(* CoDeSys 2.3.9.40 project: doz_qizil.pro *)
(* Libraries: STANDARD.LIB 4.10.05 11:14:46, IECSFC.LIB 13.4.06 15:51:28, SYSLIBTIME.LIB 20.2.06 13:31:16, SYSTASKINFO.LIB 20.2.06 13:31:38, ANALYZATION.LIB 5.10.99 09:05:06, SYSLIBCALLBACK.LIB 20.2.06 13:31:08, Util.lib 18.5.10 15:14:28 *)

(* PLC configuration (modules and I/O channels)
Fast discrete inputs [I_SIMPLE_INPUT] node 0, in %IB0 out %QB0 {Filtrationtime = 10}
  speedImpuls1 AT %IX0.0 [BitInput] Discrete input 1
  speedImpuls2 AT %IX0.1 [BitInput] Discrete input 2
  speedImpuls3 AT %IX0.2 [BitInput] Discrete input 3
  speedImpuls4 AT %IX0.3 [BitInput] Discrete input 4
AT %IB1.0 [ByteInput] 8 discrete inputs
AT %IB1.1 [ByteInput] 8 discrete inputs
AT %IB1.2 [ByteInput] 8 discrete inputs
AT %IB1.3 [ByteInput] 8 discrete inputs
Fast discrete outputs [OWEN_ID570] node 2, in %IB2 out %QB2 {SafeValueBool = FALSE; SafeValueBool = FALSE; SafeValueBool = FALSE; SafeValueBool = FALSE; Visibility = No}
  runChastot1 AT %QX2.0 [BitOutput] Fast discrete output 1
  runChastot2 AT %QX2.1 [BitOutput] Fast discrete output 2
  runChastot3 AT %QX2.2 [BitOutput] Fast discrete output 3
  runChastot4 AT %QX2.3 [BitOutput] Fast discrete output 4
Discrete outputs [ID131] node 3, in %IB3 out %QB3 {SafeValueByte = 0; SafeValueByte = 0; SafeValueByteM = 0; Visibility = No; PinCount = 24}
  AT %QB3.0 [ByteOutput] 8 discrete outputs
  AT %QB3.1 [ByteOutput] 8 discrete outputs
  AT %QB3.2 [ByteOutput] 4 discrete outputs
Special input [ID103] node 4, in %IB4 out %QB4 {Filtrationtime = 1000; PinCount = 1; WatchDogPeriod = 400; PollPeriod = 3000; Visibility = No}
  AT %IX4.0 [BitInput] Special input
Special output [ID104] node 5, in %IB5 out %QB5 {Visibility = No; PinCount = 1}
  AT %QX5.0 [BitOutput] Special output
DCON (Master) [DCON_MASTER_ID452] node 6, in %IB6 out %QB6 {Visibility = No}
  AT %QW6.0 [WordOutput] Last error
  RS-485-1 [COM1_USART] node 0, in %IB6.0 out %QB6.0 {CommunicationSpeed = 57600; Parity = NO PARITY CHECK; BitLength = 8 bits; StopLength = One stop bit; InterfaceType = RS485; FrameOriented = ASCII; Timeout = 0; Visibility = No}
  Universal DCON device [ID2100] node 1, in %IB6.1 out %QB6.1 {ReqFormat = #010[7s]; GoodResponseFormat = [1s]; BadResponseFormat = ?; ServiceTimeout = 150; RequestType = By poll time; PeriodOfService = 100; Visibility = No}
    AT %QW6.1.0 [WordOutput] Status
AT %IB6.1.0.0 [StringInput]
outVolt1 AT %QB6.1.1.0 [StringOutput]
Universal DCON device [ID2100] node 2, in %IB6.2 out %QB6.2 {ReqFormat = #011[7s]; GoodResponseFormat = [1s]; BadResponseFormat = ?; ServiceTimeout = 150; RequestType = By poll time; PeriodOfService = 100; Visibility = No}
  AT %QW6.2.0 [WordOutput] Status
AT %IB6.2.0.0 [StringInput]
outVolt2 AT %QB6.2.1.0 [StringOutput]
Universal DCON device [ID2100] node 3, in %IB6.3 out %QB6.3 {ReqFormat = #012[7s]; GoodResponseFormat = [1s]; BadResponseFormat = ?; ServiceTimeout = 150; RequestType = By poll time; PeriodOfService = 100; Visibility = No}
  AT %QW6.3.0 [WordOutput] Status
AT %IB6.3.0.0 [StringInput]
outVolt3 AT %QB6.3.1.0 [StringOutput]
Universal DCON device [ID2100] node 4, in %IB6.4 out %QB6.4 {ReqFormat = #013[7s]; GoodResponseFormat = [1s]; BadResponseFormat = ?; ServiceTimeout = 150; RequestType = By poll time; PeriodOfService = 100; Visibility = No}
  AT %QW6.4.0 [WordOutput] Status
AT %IB6.4.0.0 [StringInput]
outVolt4 AT %QB6.4.1.0 [StringOutput]
Universal DCON device [ID2100] node 5, in %IB6.5 out %QB6.5 {ReqFormat = #021; GoodResponseFormat = >[7f]; BadResponseFormat = ?; ServiceTimeout = 150; RequestType = By poll time; PeriodOfService = 100; Visibility = No}
  AT %QW6.5.0 [WordOutput] Status
dozWeight1 AT %ID6.5.0.0 [FloatInput]
Universal DCON device [ID2100] node 6, in %IB6.6 out %QB6.6 {ReqFormat = #022; GoodResponseFormat = >[7f]; BadResponseFormat = ?; ServiceTimeout = 150; RequestType = By poll time; PeriodOfService = 100; Visibility = No}
  AT %QW6.6.0 [WordOutput] Status
dozWeight2 AT %ID6.6.0.0 [FloatInput]
Universal DCON device [ID2100] node 7, in %IB6.7 out %QB6.7 {ReqFormat = #023; GoodResponseFormat = >[7f]; BadResponseFormat = ?; ServiceTimeout = 150; RequestType = By poll time; PeriodOfService = 100; Visibility = No}
  AT %QW6.7.0 [WordOutput] Status
dozWeight3 AT %ID6.7.0.0 [FloatInput]
Universal DCON device [ID2100] node 8, in %IB6.8 out %QB6.8 {ReqFormat = #024; GoodResponseFormat = >[7f]; BadResponseFormat = ?; ServiceTimeout = 150; RequestType = By poll time; PeriodOfService = 100; Visibility = No}
  AT %QW6.8.0 [WordOutput] Status
dozWeight4 AT %ID6.8.0.0 [FloatInput]
RS-232 [COM2_USART] node 0, in %IB7.0.0 out %QB7.0.0 {CommunicationSpeed = 57600; Parity = NO PARITY CHECK; BitLength = 8 bits; StopLength = One stop bit; InterfaceType = RS232; FrameOriented = RTU; Timeout = 0; Visibility = No}
Debug RS-232 [DEBUG_USART] node 1, in %IB7.0.1 out %QB7.0.1 {CommunicationSpeed = 57600; Parity = NO PARITY CHECK; BitLength = 8 bits; StopLength = One stop bit; InterfaceType = RS232; FrameOriented = RTU; Timeout = 0; Visibility = No}
AT %QD7.1.0 [FloatOutput]
AT %QD7.2.0 [FloatOutput]
AT %QD7.3.0 [FloatOutput]
AT %QD7.4.0 [FloatOutput]
AT %QD7.5.0 [FloatOutput]
AT %QD7.6.0 [FloatOutput]
AT %QD7.7.0 [FloatOutput]
AT %QD7.8.0 [FloatOutput]
AT %QD7.9.0 [FloatOutput]
AT %QD7.10.0 [FloatOutput]
AT %QD7.11.0 [FloatOutput]
AT %QD7.12.0 [FloatOutput]
AT %QD7.13.0 [FloatOutput]
AT %QD7.14.0 [FloatOutput]
AT %QD7.15.0 [FloatOutput]
AT %QD7.16.0 [FloatOutput]
AT %QD7.17.0 [FloatOutput]
AT %QD7.18.0 [FloatOutput]
AT %QD7.19.0 [FloatOutput]
AT %QD7.20.0 [FloatOutput]
AT %QD7.21.0 [FloatOutput]
AT %QD7.22.0 [FloatOutput]
AT %QD7.23.0 [FloatOutput]
AT %QD7.24.0 [FloatOutput]
AT %QD7.25.0 [FloatOutput]
AT %QD7.26.0 [FloatOutput]
AT %QD7.27.0 [FloatOutput]
AT %QD7.28.0 [FloatOutput]
AT %QD7.29.0 [FloatOutput]
AT %QD7.30.0 [FloatOutput]
AT %QD7.31.0 [FloatOutput]
AT %QD7.32.0 [FloatOutput]
AT %QD7.33.0 [FloatOutput]
AT %QD7.34.0 [FloatOutput]
AT %QD7.35.0 [FloatOutput]
AT %QD7.36.0 [FloatOutput]
AT %QD7.37.0 [FloatOutput]
AT %QD7.38.0 [FloatOutput]
AT %QD7.39.0 [FloatOutput]
AT %QD7.40.0 [FloatOutput]
AT %QD7.41.0 [FloatOutput]
AT %QW7.42.0 [WordOutput]
AT %QW7.43.0 [WordOutput]
AT %QW7.44.0 [WordOutput]
AT %QW7.45.0 [WordOutput]
8 bits [8Bit] node 46, in %IB7.46 out %QB7.46
  AT %QB7.46.0 [ByteOutput]
8 bits [8Bit] node 47, in %IB7.47 out %QB7.47
  AT %QB7.47.0 [ByteOutput]
8 bits [8Bit] node 48, in %IB7.48 out %QB7.48
  AT %QB7.48.0 [ByteOutput]
  AT %QB7.49.0 [ByteOutput]
Float [Float] node 50, in %IB7.50 out %QB7.50
  AT %QD7.50.0 [FloatOutput]
  AT %QD7.51.0 [FloatOutput]
  AT %QD7.52.0 [FloatOutput]
  AT %QD7.53.0 [FloatOutput]
  AT %QD7.54.0 [FloatOutput]
  AT %QD7.55.0 [FloatOutput]
  AT %QD7.56.0 [FloatOutput]
  AT %QD7.57.0 [FloatOutput]
  AT %QD7.58.0 [FloatOutput]
  AT %QD7.59.0 [FloatOutput]
Float [Float] node 60, in %IB7.60 out %QB7.60
  AT %QD7.60.0 [FloatOutput]
2 byte [Register] node 61, in %IB7.61 out %QB7.61
  year AT %QW7.61.0 [WordOutput]
2 byte [Register] node 62, in %IB7.62 out %QB7.62
  month AT %QW7.62.0 [WordOutput]
2 byte [Register] node 63, in %IB7.63 out %QB7.63
  day AT %QW7.63.0 [WordOutput]
2 byte [Register] node 64, in %IB7.64 out %QB7.64
  hour AT %QW7.64.0 [WordOutput]
2 byte [Register] node 65, in %IB7.65 out %QB7.65
  minute AT %QW7.65.0 [WordOutput]
2 byte [Register] node 66, in %IB7.66 out %QB7.66
  sekund AT %QW7.66.0 [WordOutput]
2 byte [Register] node 67, in %IB7.67 out %QB7.67
  taskDozSpeed1 AT %QW7.67.0 [WordOutput]
2 byte [Register] node 68, in %IB7.68 out %QB7.68
  taskDozSpeed2 AT %QW7.68.0 [WordOutput]
2 byte [Register] node 69, in %IB7.69 out %QB7.69
  taskDozSpeed3 AT %QW7.69.0 [WordOutput]
2 byte [Register] node 70, in %IB7.70 out %QB7.70
  taskDozSpeed4 AT %QW7.70.0 [WordOutput]
  workMode AT %QW7.71.0 [WordOutput]
  AT %QW7.72.0 [WordOutput]
taraSpeedDoz1 AT %QD7.73.0 [FloatOutput]
taraSpeedDoz2 AT %QD7.74.0 [FloatOutput]
taraSpeedDoz3 AT %QD7.75.0 [FloatOutput]
taraSpeedDoz4 AT %QD7.76.0 [FloatOutput]
taraVesDoz1 AT %QD7.77.0 [FloatOutput]
taraVesDoz2 AT %QD7.78.0 [FloatOutput]
taraVesDoz3 AT %QD7.79.0 [FloatOutput]
taraVesDoz4 AT %QD7.80.0 [FloatOutput]
AT %QB7.81.0 [ByteOutput]
AT %QB7.82.0 [ByteOutput]
AT %QB7.83.0 [ByteOutput]
AT %QB7.84.0 [ByteOutput]
AT %QB7.85.0 [ByteOutput]
AT %QB7.86.0 [ByteOutput]
AT %QB7.87.0 [ByteOutput]
AT %QB7.88.0 [ByteOutput]
ModBus (Master) [MODBUS_MASTER_ID450] node 8, in %IB8 out %QB8 {Visibility = No}
  AT %QD8.0 [DWordOutput] Last address
  AT %QW8.1 [WordOutput] Last error
  RS-485-2 [COM3_USART] node 0, in %IB8.0 out %QB8.0 {CommunicationSpeed = 11520; Parity = NO PARITY CHECK; BitLength = 8 bits; StopLength = One stop bit; InterfaceType = RS485; FrameOriented = RTU; Timeout = 0; Visibility = No}
AT %QB8.1.0 [ComChannel] Command (0xff - Start)
freqStatus1 AT %IW8.1.0.0 [WordInput]
freqChastot1 AT %IW8.1.1.0 [WordInput]
freqChastotZadan1 AT %IW8.1.2.0 [WordInput]
freqTok1 AT %IW8.1.3.0 [WordInput]
AT %QB8.2.0 [ComChannel] Command (0xff - Start)
freqStatus2 AT %IW8.2.0.0 [WordInput]
freqChastot2 AT %IW8.2.1.0 [WordInput]
freqChastotZadan2 AT %IW8.2.2.0 [WordInput]
freqTok2 AT %IW8.2.3.0 [WordInput]
AT %QB8.3.0 [ComChannel] Command (0xff - Start)
freqStatus3 AT %IW8.3.0.0 [WordInput]
freqChastot3 AT %IW8.3.1.0 [WordInput]
freqChastotZadan3 AT %IW8.3.2.0 [WordInput]
freqTok3 AT %IW8.3.3.0 [WordInput]
AT %QB8.4.0 [ComChannel] Command (0xff - Start)
freqStatus4 AT %IW8.4.0.0 [WordInput]
freqChastot4 AT %IW8.4.1.0 [WordInput]
freqChastotZadan4 AT %IW8.4.2.0 [WordInput]
freqTok4 AT %IW8.4.3.0 [WordInput]
AT %IX9.0 [BitInput] Button Start/Stop
*)

(* Global variable list: Global_Variables *)
VAR_GLOBAL
	currProizDoz1 AT %QD7.1.0 : REAL; (* 0 *)
	currProizDoz2 AT %QD7.2.0 : REAL; (* 2 *)
	currProizDoz3 AT %QD7.3.0 : REAL; (* 4 *)
	currProizDoz4 AT %QD7.4.0 : REAL; (* 6 *)
	currProizDozTotal AT %QD7.58.0 : REAL; (* 104 *)
	(**************************************************)
	taskDozPercent1 AT %QD7.5.0 : REAL; (* 8 *)
	taskDozPercent2 AT %QD7.6.0 : REAL; (* 10 *)
	taskDozPercent3 AT %QD7.7.0 : REAL; (* 12 *)
	taskDozPercent4 AT %QD7.8.0 : REAL; (* 14 *)
	(**************************************************)
	dozCount1 AT %QD7.9.0 : REAL; (* 16 *)
	dozCount2 AT %QD7.10.0 : REAL; (* 18 *)
	dozCount3 AT %QD7.11.0 : REAL; (* 20 *)
	dozCount4 AT %QD7.12.0 : REAL; (* 22 *)
	dozCountTotal AT %QD7.59.0 : REAL; (* 106 *)
	(**************************************************)
	dozSpeed1 AT %QD7.13.0 : REAL; (* 24 *)
	dozSpeed2 AT %QD7.14.0 : REAL; (* 26 *)
	dozSpeed3 AT %QD7.15.0 : REAL; (* 28 *)
	dozSpeed4 AT %QD7.16.0 : REAL; (* 30 *)
	(**************************************************)
	dozMilliVolt1 AT %QD7.17.0 : REAL; (* 32 *)
	dozMilliVolt2 AT %QD7.18.0 : REAL; (* 34 *)
	dozMilliVolt3 AT %QD7.19.0 : REAL; (* 36 *)
	dozMilliVolt4 AT %QD7.20.0 : REAL; (* 38 *)
	(**************************************************)
	chatotTok1 AT %QD7.21.0 : REAL; (* 40 *)
	chatotTok2 AT %QD7.22.0 : REAL; (* 42 *)
	chatotTok3 AT %QD7.23.0 : REAL; (* 44 *)
	chatotTok4 AT %QD7.24.0 : REAL; (* 46 *)
	(**************************************************)
	chatotFreq1 AT %QD7.25.0 : REAL; (* 48 *)
	chatotFreq2 AT %QD7.26.0 : REAL; (* 50 *)
	chatotFreq3 AT %QD7.27.0 : REAL; (* 52 *)
	chatotFreq4 AT %QD7.28.0 : REAL; (* 54 *)
	(**************************************************)
	taskTotal AT %QD7.29.0: REAL;	(* 56 *)
	(**************************************************)
	dozKoefPerVESDoz1 AT %QD7.30.0: REAL;	(* 58 *)
	dozKoefPerVESDoz2 AT %QD7.31.0: REAL;	(* 60 *)
	dozKoefPerVESDoz3 AT %QD7.32.0 : REAL; (* 62 *)
	dozKoefPerVESDoz4 AT %QD7.33.0 : REAL; (* 64 *)
	(**************************************************)
	dozKoefSpeedDoz1 AT %QD7.34.0 : REAL; (* 66 *)
	dozKoefSpeedDoz2 AT %QD7.35.0 : REAL; (* 68 *)
	dozKoefSpeedDoz3 AT %QD7.36.0 : REAL; (* 70 *)
	dozKoefSpeedDoz4 AT %QD7.37.0 : REAL; (* 72 *)
	(**************************************************)
	dozDreyfDoz1 AT %QD7.38.0 : REAL; (* 74 *)
	dozDreyfDoz2 AT %QD7.39.0 : REAL; (* 76 *)
	dozDreyfDoz3 AT %QD7.40.0 : REAL; (* 78 *)
	dozDreyfDoz4 AT %QD7.41.0 : REAL; (* 80 *)
	(**************************************************)
	dozSkolTimeDoz1 AT %QW7.42.0 : WORD; (* 82 *)
	dozSkolTimeDoz2 AT %QW7.43.0 : WORD; (* 83 *)
	dozSkolTimeDoz3 AT %QW7.44.0 : WORD; (* 84 *)
	dozSkolTimeDoz4 AT %QW7.45.0 : WORD; (* 85 *)
	(**************************************************)
	KoefPer1 AT %QX7.46.0.0 : BOOL; (* 0008600 *)
	KoefPer2 AT %QX7.46.0.1 : BOOL; (* 0008601 *)
	KoefPer3 AT %QX7.46.0.2 : BOOL; (* 0008602 *)
	KoefPer4 AT %QX7.46.0.3 : BOOL; (* 0008603 *)
	(**************************************************)
	KoefSpeed1 AT %QX7.46.0.4 : BOOL; (* 0008604 *)
	KoefSpeed2 AT %QX7.46.0.5 : BOOL; (* 0008605 *)
	KoefSpeed3 AT %QX7.46.0.6 : BOOL; (* 0008606 *)
	KoefSpeed4 AT %QX7.46.0.7 : BOOL; (* 0008607 *)
	(**************************************************)
	dreyf1 AT %QX7.47.0.0 : BOOL; (* 0008608 *)
	dreyf2 AT %QX7.47.0.1 : BOOL; (* 0008609 *)
	dreyf3 AT %QX7.47.0.2 : BOOL; (* 0008610 *)
	dreyf4 AT %QX7.47.0.3 : BOOL; (* 0008611 *)
	(**************************************************)
	resetError AT %QX7.47.0.4 : BOOL; (* 0008612 *)
	timeSinxron AT %QX7.47.0.5 : BOOL; (* 0008613 *)
	(**************************************************)
	dozInGroup1 AT %QX7.48.0.0 : BOOL; (* 0008700 *)
	dozInGroup2 AT %QX7.48.0.1 : BOOL; (* 0008701 *)
	dozInGroup3 AT %QX7.48.0.2 : BOOL; (* 0008702 *)
	dozInGroup4 AT %QX7.48.0.3 : BOOL; (* 0008703 *)
	(**************************************************)
	dozWork1 AT %QX7.48.0.4 : BOOL; (* 0008704 *)
	dozWork2 AT %QX7.48.0.5 : BOOL; (* 0008705 *)
	dozWork3 AT %QX7.48.0.6 : BOOL; (* 0008706 *)
	dozWork4 AT %QX7.48.0.7 : BOOL; (* 0008707 *)
	(**************************************************)
	run1 AT %QX7.49.0.0 : BOOL; (* 0008708 *)
	run2 AT %QX7.49.0.1 : BOOL; (* 0008709 *)
	run3 AT %QX7.49.0.2 : BOOL; (* 0008710 *)
	run4 AT %QX7.49.0.3 : BOOL; (* 0008711 *)
	(**************************************************)
	dozWieght1 AT %QD7.50.0 : REAL; (* 88 *)
	dozWieght2 AT %QD7.51.0 : REAL; (* 90 *)
	dozWieght3 AT %QD7.52.0 : REAL; (* 92 *)
	dozWieght4 AT %QD7.53.0 : REAL; (* 94 *)
	(**************************************************)
	taskProizDoz1 AT %QD7.54.0 : REAL; (* 96 *)
	taskProizDoz2 AT %QD7.55.0 : REAL; (* 98 *)
	taskProizDoz3 AT %QD7.56.0 : REAL; (* 100 *)
	taskProizDoz4 AT %QD7.57.0 : REAL; (* 102 *)
	(**************************************************)
	dreyfTaraVes1 : REAL;
	dreyfTaraVes2 : REAL;
	dreyfTaraVes3 : REAL;
	dreyfTaraVes4 : REAL;

END_VAR

(* POU PLC_PRG, ST *)
PROGRAM PLC_PRG
VAR
	temp : WORD;
END_VAR
(*****************************)
translate();
errors();
sinxron();
sirenStart();
sirenStop();
stopCFC();
(*****************************)
IF(temp <> workMode) THEN
	stopCFC();
	temp := workMode;
END_IF;

CASE workMode OF
	11 : taraSpeedModeDoz1();
	12 : taraSpeedModeDoz2();
	13 : taraSpeedModeDoz3();
	14 : taraSpeedModeDoz4();
	21 : taraVesModeDoz1();
	22 : taraVesModeDoz2();
	23 : taraVesModeDoz3();
	24 : taraVesModeDoz4();
ELSE
	 auto ();
END_CASE;
END_PROGRAM

(* POU translate, ST *)
PROGRAM translate
VAR
	count1 : HISOBLAGICH;
	count2 : HISOBLAGICH;
	count3 : HISOBLAGICH;
	count4 : HISOBLAGICH;

	calcWeight1 : CALCWEIGHT;
	calcWeight2 : CALCWEIGHT;
	calcWeight3 : CALCWEIGHT;
	calcWeight4 : CALCWEIGHT;

	filtr1 : ANALOGFILTR;
	filtr2 : ANALOGFILTR;
	filtr3 : ANALOGFILTR;
	filtr4 : ANALOGFILTR;




END_VAR
(**************************************************)
count1(	tezlik := dozSpeed1,
			proizvodMgn := currProizDoz1,
			SUMMA => dozCount1);
count2(tezlik := dozSpeed2,
			proizvodMgn := currProizDoz2,
			SUMMA => dozCount2);
count3(	tezlik := dozSpeed3,
			proizvodMgn := currProizDoz3,
			SUMMA => dozCount3);
count4(tezlik := dozSpeed4,
			proizvodMgn := currProizDoz4,
			SUMMA => dozCount4);
dozSpeed1 := dozKoefSpeedDoz1 * freqChastotZadan1 ;
dozSpeed2 := dozKoefSpeedDoz2 * freqChastotZadan2;
dozSpeed3 := dozKoefSpeedDoz3 * freqChastotZadan3;
dozSpeed4 := dozKoefSpeedDoz4 * freqChastotZadan4;

calcWeight1(dreyfNol := dozDreyfDoz1,
				koeffitsentPeredachaVes := dozKoefPerVESDoz1,
				milliVolt := dozMilliVolt1,
				Ves => dozWieght2);
calcWeight2(dreyfNol := dozDreyfDoz2,
				koeffitsentPeredachaVes := dozKoefPerVESDoz2,
				milliVolt := dozMilliVolt2,
				Ves => dozWieght2);
calcWeight3(dreyfNol := dozDreyfDoz3,
				koeffitsentPeredachaVes := dozKoefPerVESDoz3,
				milliVolt := dozMilliVolt3,
				Ves => dozWieght3);
calcWeight4(dreyfNol := dozDreyfDoz4,
				koeffitsentPeredachaVes := dozKoefPerVESDoz4,
				milliVolt := dozMilliVolt4,
				Ves => dozWieght4);

dozInGroup1 := doz1InGroup;
dozInGroup2 := doz2InGroup;
dozInGroup3 := doz3InGroup;
dozInGroup4 := doz4InGroup;
currProizDozTotal := currProizDoz1 + currProizDoz2 + currProizDoz3 + currProizDoz4;
dozCountTotal := dozCount1 + dozCount2 + dozCount3 + dozCount4;
(***********************************************)
taskProizDoz1 := taskTotal * taskDozPercent1/100;
taskProizDoz2 := taskTotal * taskDozPercent2/100;
taskProizDoz3 := taskTotal * taskDozPercent3/100;
taskProizDoz4 := taskTotal * taskDozPercent4/100;
(********************************************)
dozWork1 := freqStatus1.0 AND freqStatus1.1;
dozWork2 := freqStatus2.0 AND freqStatus2.1;
dozWork3 := freqStatus3.0 AND freqStatus3.1;
dozWork4 := freqStatus4.0 AND freqStatus4.1;
(********************************************)
chatotTok1 := WORD_TO_REAL(freqTok1)/100;
chatotTok2 := WORD_TO_REAL(freqTok2)/100;
chatotTok3 := WORD_TO_REAL(freqTok3)/100;
chatotTok4 := WORD_TO_REAL(freqTok4)/100;
(*********************************************)
chatotFreq1 := WORD_TO_REAL(freqChastot1)/100;
chatotFreq2 := WORD_TO_REAL(freqChastot2)/100;
chatotFreq3 := WORD_TO_REAL(freqChastot3)/100;
chatotFreq4 := WORD_TO_REAL(freqChastot4)/100;
(*********************************************)
IF(dozAuto1 = FALSE) THEN
	taskDozPercent1 := (currProizDoz1 / taskTotal) * 100 ;
END_IF;
IF(dozAuto2 = FALSE) THEN
	taskDozPercent2 := (currProizDoz2 / taskTotal) * 100 ;
END_IF;
IF(dozAuto3 = FALSE) THEN
	taskDozPercent3 := (currProizDoz3 / taskTotal) * 100 ;
END_IF;
IF(dozAuto4 = FALSE) THEN
	taskDozPercent4 := (currProizDoz4 / taskTotal) * 100 ;
END_IF;
(*********************************************)

(***********************************************)

filtr1(inputAnalog := dozWeight1, vaqt := 1000, analogResult => dozMilliVolt1);
filtr2(inputAnalog := dozWeight2, vaqt := 1000, analogResult => dozMilliVolt2);
filtr3(inputAnalog := dozWeight3, vaqt := 1000, analogResult => dozMilliVolt3);
filtr4(inputAnalog := dozWeight4, vaqt := 1000, analogResult => dozMilliVolt4);
(*
dozMilliVolt1 := dozWeight1;
dozMilliVolt2 := dozWeight2;
dozMilliVolt3 := dozWeight3;
dozMilliVolt4 := dozWeight4;
*)
dozWieght1 := (dozMilliVolt1 - dozDreyfDoz1) * dozKoefPerVESDoz1;
dozWieght2 := (dozMilliVolt2 - dozDreyfDoz2) * dozKoefPerVESDoz2;
dozWieght3 := (dozMilliVolt3 - dozDreyfDoz3) * dozKoefPerVESDoz3;
dozWieght4 := (dozMilliVolt4 - dozDreyfDoz4) * dozKoefPerVESDoz4;

(********************************************)
currProizDoz1 := dozWieght1 * (dozSpeed1 * 3600.0) / 100000;
currProizDoz2 := dozWieght2 * (dozSpeed2 * 3600.0) / 100000;
currProizDoz3 := dozWieght3 * (dozSpeed3 * 3600.0) / 100000;
currProizDoz4 := dozWieght4 * (dozSpeed4 * 3600.0) / 100000;
END_PROGRAM

(* POU HISOBLAGICH, ST *)
FUNCTION_BLOCK HISOBLAGICH
VAR_INPUT
	proizvodMgn : REAL;  (* Dozatorning ishlab chiqarish quvvati *)
	tezlik : REAL;		  (* Dozatorni tezligi *)
END_VAR
VAR_OUTPUT
	SUMMA : REAL; (* Jami o'tkazilgan mahsulot *)
END_VAR
VAR
	tmrCount: TON;
END_VAR
IF(tezlik > 0) THEN
	tmrCount(IN := TRUE, PT := T#1s);
	IF(tmrCount.Q = TRUE) THEN
		SUMMA := SUMMA + proizvodMgn / 3600;
		tmrCount(IN := FALSE);
	END_IF;
END_IF;
END_FUNCTION_BLOCK

(* POU CALCWEIGHT, CFC *)
FUNCTION_BLOCK CALCWEIGHT
VAR_INPUT
	milliVolt: REAL; 	(*Tenzo datchikdan keladigan millivolt*)
	dreyfNol: REAL; 	(*Tenzo datchikni usti bo'sh turgandagi millivolt*)
	koeffitsentPeredachaVes: REAL;	(*Koeffitsent peredacha ves na pogon metr*)
END_VAR
VAR_OUTPUT
	Ves: REAL;		(*Tenzo datchik o'lchgandan keyingi tayyor yuk kg da*)
END_VAR
VAR
END_VAR
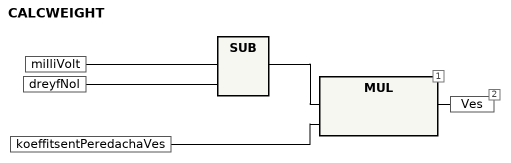
_CFC_ (* Continuous Function Chart, elements in execution order *)
#0 SUB(milliVolt, dreyfNol)
#1 MUL(#0, koeffitsentPeredachaVes)
#2 Ves <= #1
_END_CFC_
(* the same logic as Structured Text *)
Ves := (milliVolt - dreyfNol) * koeffitsentPeredachaVes;
END_FUNCTION_BLOCK

(* POU ANALOGFILTR, ST *)
FUNCTION_BLOCK ANALOGFILTR
VAR_INPUT
	vaqt : WORD := 1000;
	inputAnalog : REAL;
END_VAR
VAR_OUTPUT
	analogResult : REAL;
END_VAR
VAR
	tmr_f: TON;
	sumAnalog : REAL;
	countOfanalog : DWORD;
END_VAR
tmr_f(IN := TRUE, PT := T#1ms * vaqt);
IF(tmr_f.Q = TRUE) THEN
	analogResult := sumAnalog / countOfanalog;
	sumAnalog := 0;
	countOfanalog := 1;
	tmr_f(IN := FALSE);
ELSE
	sumAnalog := sumAnalog + inputAnalog;
	countOfanalog := countOfanalog + 1;

END_IF;
END_FUNCTION_BLOCK

(* POU errors, CFC *)
PROGRAM errors
VAR
	YUK: REAL := 2.5;
	trig_weight2: R_TRIG;
	trig_weight1: R_TRIG;
	trigReset: R_TRIG;
	trig_weight3: R_TRIG;
	trig_weight4: R_TRIG;
	tonWeight4: TON;
	vaqt : TIME := T#10S;
	tonWeight1: TON;
	tonWeight2: TON;
	tonWeight3: TON;
(********************************)
	trig_igroupR1: R_TRIG;
	trig_igroupF1: F_TRIG;
	trig_igroupR2: R_TRIG;
	trig_igroupF2: F_TRIG;
	trig_igroupR3: R_TRIG;
	trig_igroupF3: F_TRIG;
	trig_igroupR4: R_TRIG;
	trig_igroupF4: F_TRIG;
	trig_slideR1: R_TRIG;
	trig_slideF1: F_TRIG;
	(*************************************)
	tonslide1: TON;

END_VAR
VAR (* helpers for the ST form of the networks *)
	_t80 : BOOL;
	_t137 : BOOL;
	_t158 : BOOL;
	_en155 : BOOL;
	_t155 : BOOL;
	_t136 : BOOL;
	_t1 : BOOL;
	_t180 : BOOL;
	_t174 : BOOL;
	_en178 : BOOL;
	_t178 : BOOL;
	_t183 : BOOL;
	_t199 : BOOL;
	_t193 : BOOL;
	_en197 : BOOL;
	_t197 : BOOL;
	_t202 : BOOL;
	_t218 : BOOL;
	_t212 : BOOL;
	_en216 : BOOL;
	_t216 : BOOL;
	_t221 : BOOL;
END_VAR
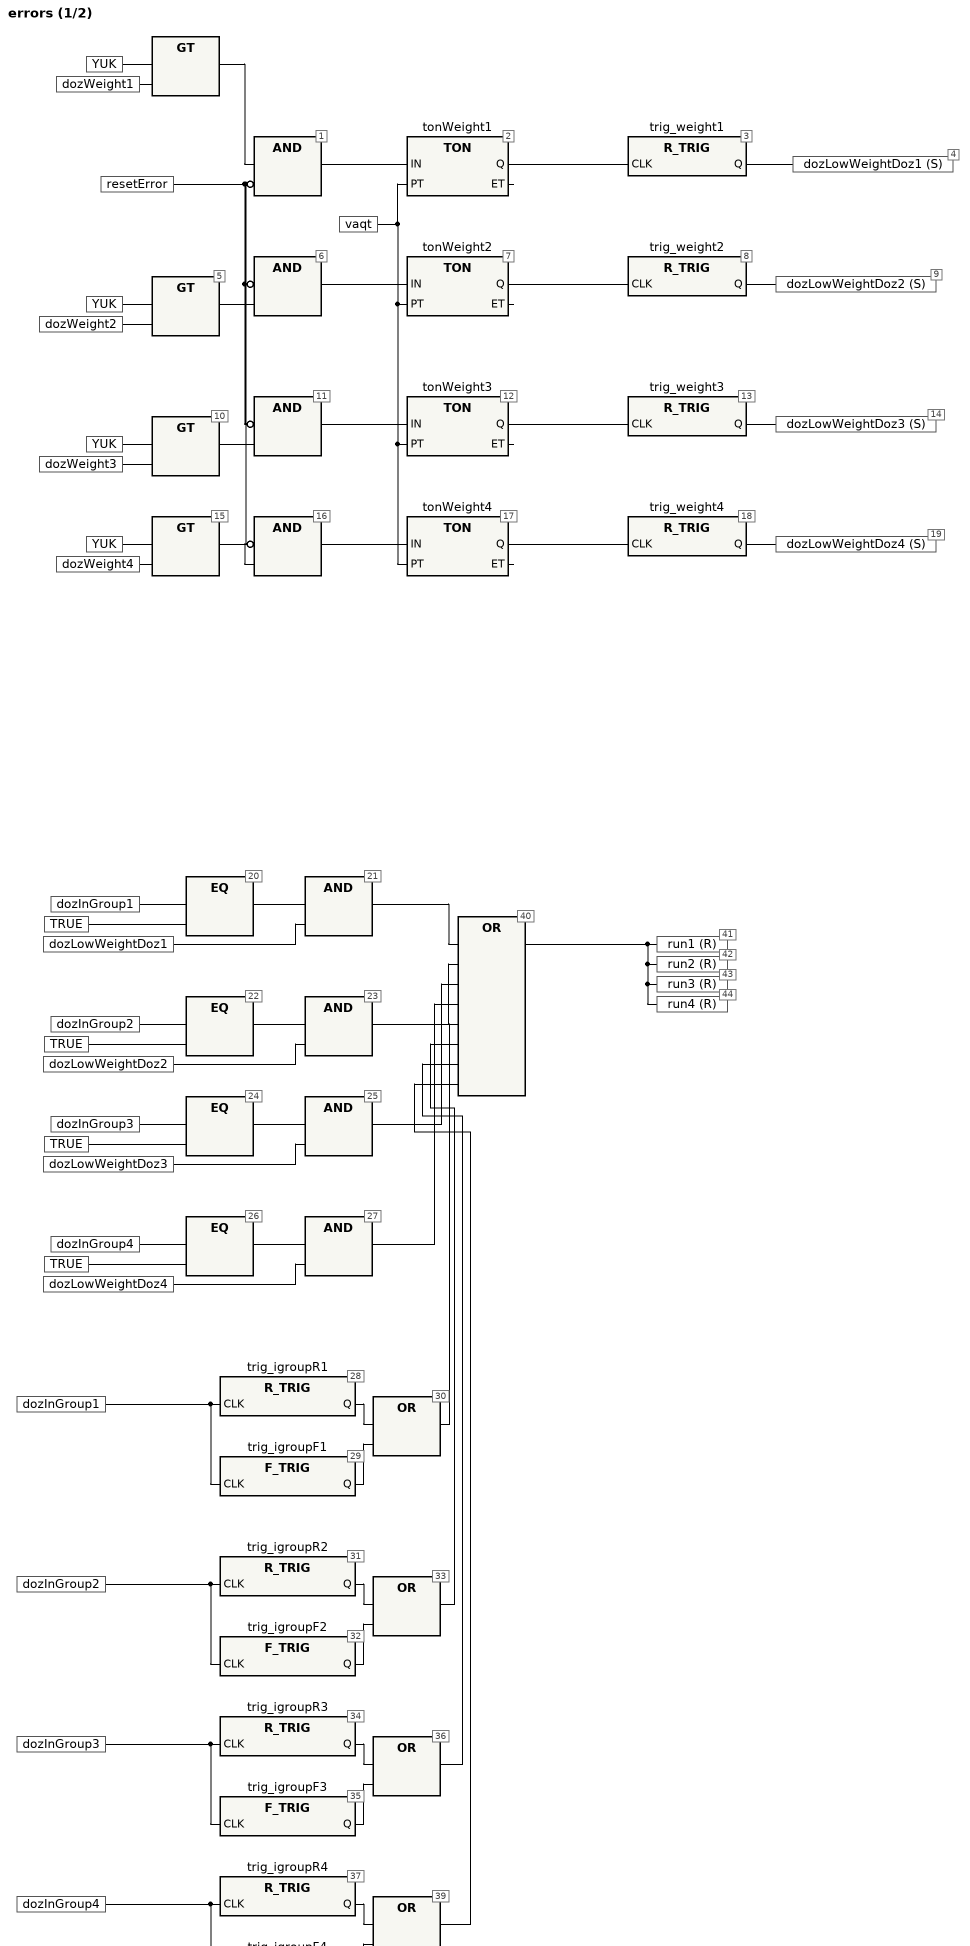
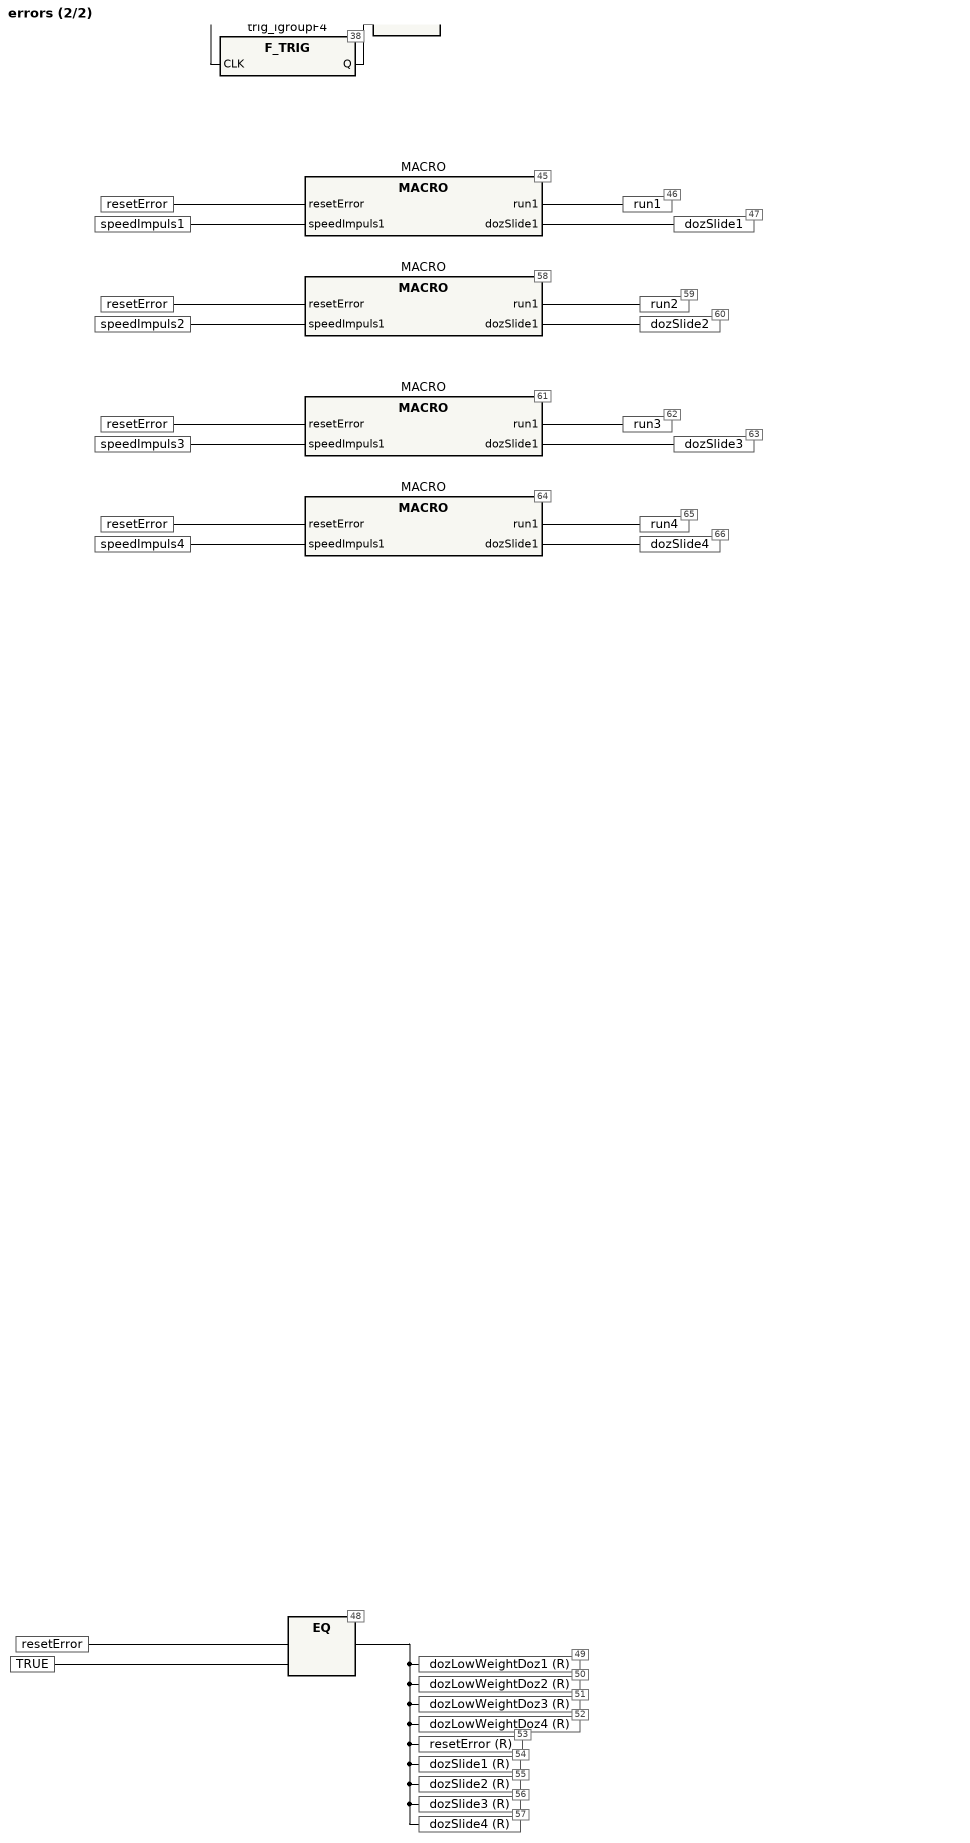
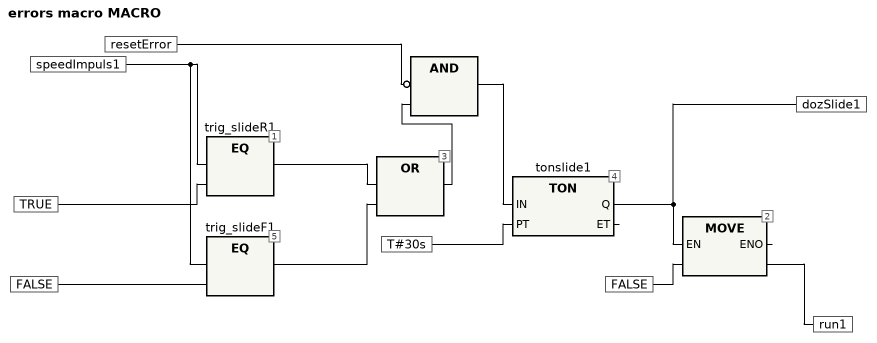
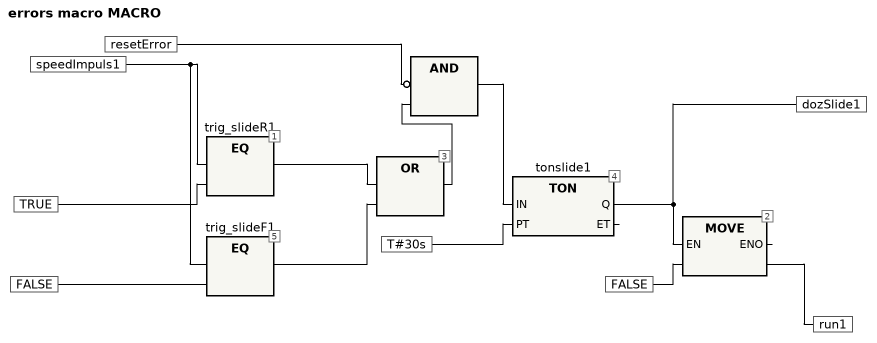
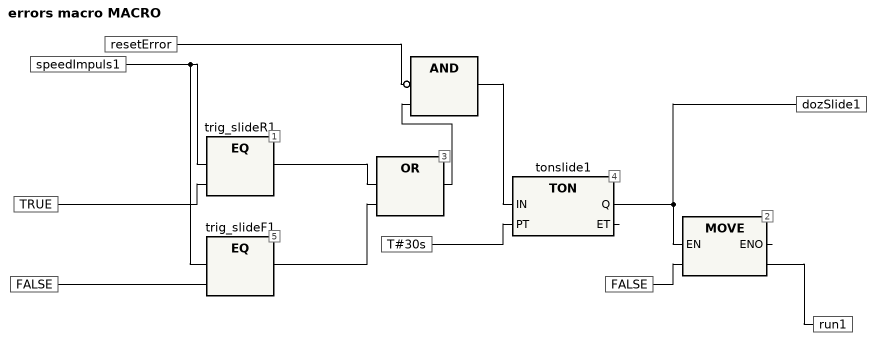
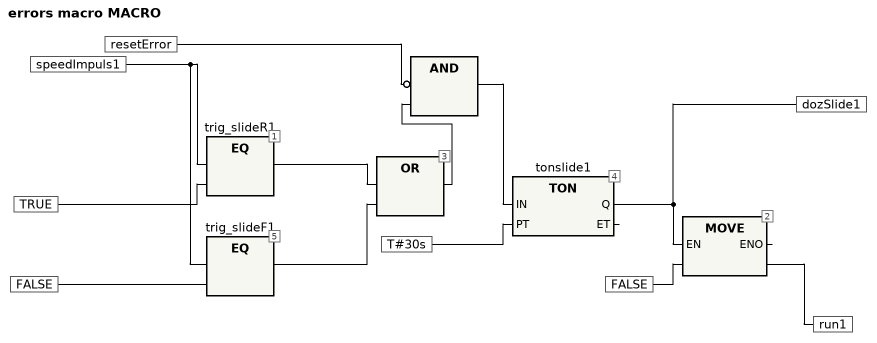
_CFC_ (* Continuous Function Chart, elements in execution order *)
#0 GT(YUK, dozWeight1)
#1 AND(#0, NOT resetError)
#2 tonWeight1:TON(IN: #1, PT: vaqt)
#3 trig_weight1:R_TRIG(CLK: #2.Q)
#4 S dozLowWeightDoz1 <= #3.Q
#5 GT(YUK, dozWeight2)
#6 AND(NOT resetError, #5)
#7 tonWeight2:TON(IN: #6, PT: vaqt)
#8 trig_weight2:R_TRIG(CLK: #7.Q)
#9 S dozLowWeightDoz2 <= #8.Q
#10 GT(YUK, dozWeight3)
#11 AND(NOT resetError, #10)
#12 tonWeight3:TON(IN: #11, PT: vaqt)
#13 trig_weight3:R_TRIG(CLK: #12.Q)
#14 S dozLowWeightDoz3 <= #13.Q
#15 GT(YUK, dozWeight4)
#16 AND(NOT resetError, #15)
#17 tonWeight4:TON(IN: #16, PT: vaqt)
#18 trig_weight4:R_TRIG(CLK: #17.Q)
#19 S dozLowWeightDoz4 <= #18.Q
#20 EQ(dozInGroup1, TRUE)
#21 AND(#20, dozLowWeightDoz1)
#22 EQ(dozInGroup2, TRUE)
#23 AND(#22, dozLowWeightDoz2)
#24 EQ(dozInGroup3, TRUE)
#25 AND(#24, dozLowWeightDoz3)
#26 EQ(dozInGroup4, TRUE)
#27 AND(#26, dozLowWeightDoz4)
#28 trig_igroupR1:R_TRIG(CLK: dozInGroup1)
#29 trig_igroupF1:F_TRIG(CLK: dozInGroup1)
#30 OR(#28.Q, #29.Q)
#31 trig_igroupR2:R_TRIG(CLK: dozInGroup2)
#32 trig_igroupF2:F_TRIG(CLK: dozInGroup2)
#33 OR(#31.Q, #32.Q)
#34 trig_igroupR3:R_TRIG(CLK: dozInGroup3)
#35 trig_igroupF3:F_TRIG(CLK: dozInGroup3)
#36 OR(#34.Q, #35.Q)
#37 trig_igroupR4:R_TRIG(CLK: dozInGroup4)
#38 trig_igroupF4:F_TRIG(CLK: dozInGroup4)
#39 OR(#37.Q, #38.Q)
#40 OR(#21, #23, #25, #27, #30, #33, #36, #39)
#41 R run1 <= #40
#42 R run2 <= #40
#43 R run3 <= #40
#44 R run4 <= #40
#45 MACRO MACRO(pin 1 "resetError": resetError, pin 2 "speedImpuls1": speedImpuls1)
	#46 AND(NOT pin 1, #49)
	#47 trig_slideR1:EQ(pin 2, TRUE)
	#48 MOVE(EN: #50.Q, FALSE)
	#49 OR(#47, #51)
	#50 tonslide1:TON(IN: #46, PT: T#30s)
	#51 trig_slideF1:EQ(pin 2, FALSE)
	out 1 "run1" <= #48
	out 2 "dozSlide1" <= #50.Q
END_MACRO
#52 run1 <= #45.out 1
#53 dozSlide1 <= #45.out 2
#54 EQ(resetError, TRUE)
#55 R dozLowWeightDoz1 <= #54
#56 R dozLowWeightDoz2 <= #54
#57 R dozLowWeightDoz3 <= #54
#58 R dozLowWeightDoz4 <= #54
#59 R resetError <= #54
#60 R dozSlide1 <= #54
#61 R dozSlide2 <= #54
#62 R dozSlide3 <= #54
#63 R dozSlide4 <= #54
#64 MACRO MACRO(pin 1 "resetError": resetError, pin 2 "speedImpuls1": speedImpuls2)
	#65 AND(NOT pin 1, #68)
	#66 trig_slideR1:EQ(pin 2, TRUE)
	#67 MOVE(EN: #69.Q, FALSE)
	#68 OR(#66, #70)
	#69 tonslide1:TON(IN: #65, PT: T#30s)
	#70 trig_slideF1:EQ(pin 2, FALSE)
	out 1 "run1" <= #67
	out 2 "dozSlide1" <= #69.Q
END_MACRO
#71 run2 <= #64.out 1
#72 dozSlide2 <= #64.out 2
#73 MACRO MACRO(pin 1 "resetError": resetError, pin 2 "speedImpuls1": speedImpuls3)
	#74 AND(NOT pin 1, #77)
	#75 trig_slideR1:EQ(pin 2, TRUE)
	#76 MOVE(EN: #78.Q, FALSE)
	#77 OR(#75, #79)
	#78 tonslide1:TON(IN: #74, PT: T#30s)
	#79 trig_slideF1:EQ(pin 2, FALSE)
	out 1 "run1" <= #76
	out 2 "dozSlide1" <= #78.Q
END_MACRO
#80 run3 <= #73.out 1
#81 dozSlide3 <= #73.out 2
#82 MACRO MACRO(pin 1 "resetError": resetError, pin 2 "speedImpuls1": speedImpuls4)
	#83 AND(NOT pin 1, #86)
	#84 trig_slideR1:EQ(pin 2, TRUE)
	#85 MOVE(EN: #87.Q, FALSE)
	#86 OR(#84, #88)
	#87 tonslide1:TON(IN: #83, PT: T#30s)
	#88 trig_slideF1:EQ(pin 2, FALSE)
	out 1 "run1" <= #85
	out 2 "dozSlide1" <= #87.Q
END_MACRO
#89 run4 <= #82.out 1
#90 dozSlide4 <= #82.out 2
_END_CFC_
(* the same logic as Structured Text *)
tonWeight1(IN := (YUK > dozWeight1) AND NOT resetError, PT := vaqt);
trig_weight1(CLK := tonWeight1.Q);
IF trig_weight1.Q THEN dozLowWeightDoz1 := TRUE; END_IF;
tonWeight2(IN := NOT resetError AND (YUK > dozWeight2), PT := vaqt);
trig_weight2(CLK := tonWeight2.Q);
IF trig_weight2.Q THEN dozLowWeightDoz2 := TRUE; END_IF;
tonWeight3(IN := NOT resetError AND (YUK > dozWeight3), PT := vaqt);
trig_weight3(CLK := tonWeight3.Q);
IF trig_weight3.Q THEN dozLowWeightDoz3 := TRUE; END_IF;
tonWeight4(IN := NOT resetError AND (YUK > dozWeight4), PT := vaqt);
trig_weight4(CLK := tonWeight4.Q);
IF trig_weight4.Q THEN dozLowWeightDoz4 := TRUE; END_IF;
trig_igroupR1(CLK := dozInGroup1);
trig_igroupF1(CLK := dozInGroup1);
trig_igroupR2(CLK := dozInGroup2);
trig_igroupF2(CLK := dozInGroup2);
trig_igroupR3(CLK := dozInGroup3);
trig_igroupF3(CLK := dozInGroup3);
trig_igroupR4(CLK := dozInGroup4);
trig_igroupF4(CLK := dozInGroup4);
_t80 := ((dozInGroup1 = TRUE) AND dozLowWeightDoz1) OR ((dozInGroup2 = TRUE) AND dozLowWeightDoz2) OR ((dozInGroup3 = TRUE) AND dozLowWeightDoz3) OR ((dozInGroup4 = TRUE) AND dozLowWeightDoz4) OR (trig_igroupR1.Q OR trig_igroupF1.Q) OR (trig_igroupR2.Q OR trig_igroupF2.Q) OR (trig_igroupR3.Q OR trig_igroupF3.Q) OR (trig_igroupR4.Q OR trig_igroupF4.Q);
IF _t80 THEN run1 := FALSE; END_IF;
IF _t80 THEN run2 := FALSE; END_IF;
IF _t80 THEN run3 := FALSE; END_IF;
IF _t80 THEN run4 := FALSE; END_IF;
(* macro MACRO *)
_t158 := NOT resetError AND _t137;
_en155 := tonslide1.Q;
IF _en155 THEN _t155 := FALSE; END_IF;
_t137 := (speedImpuls1 = TRUE) OR _t136;
tonslide1(IN := _t158, PT := T#30s);
_t136 := speedImpuls1 = FALSE;
IF _en155 THEN run1 := _t155; END_IF;
dozSlide1 := tonslide1.Q;
_t1 := resetError = TRUE;
IF _t1 THEN dozLowWeightDoz1 := FALSE; END_IF;
IF _t1 THEN dozLowWeightDoz2 := FALSE; END_IF;
IF _t1 THEN dozLowWeightDoz3 := FALSE; END_IF;
IF _t1 THEN dozLowWeightDoz4 := FALSE; END_IF;
IF _t1 THEN resetError := FALSE; END_IF;
IF _t1 THEN dozSlide1 := FALSE; END_IF;
IF _t1 THEN dozSlide2 := FALSE; END_IF;
IF _t1 THEN dozSlide3 := FALSE; END_IF;
IF _t1 THEN dozSlide4 := FALSE; END_IF;
(* macro MACRO *)
_t174 := NOT resetError AND _t180;
_en178 := tonslide1.Q;
IF _en178 THEN _t178 := FALSE; END_IF;
_t180 := (speedImpuls2 = TRUE) OR _t183;
tonslide1(IN := _t174, PT := T#30s);
_t183 := speedImpuls2 = FALSE;
IF _en178 THEN run2 := _t178; END_IF;
dozSlide2 := tonslide1.Q;
(* macro MACRO *)
_t193 := NOT resetError AND _t199;
_en197 := tonslide1.Q;
IF _en197 THEN _t197 := FALSE; END_IF;
_t199 := (speedImpuls3 = TRUE) OR _t202;
tonslide1(IN := _t193, PT := T#30s);
_t202 := speedImpuls3 = FALSE;
IF _en197 THEN run3 := _t197; END_IF;
dozSlide3 := tonslide1.Q;
(* macro MACRO *)
_t212 := NOT resetError AND _t218;
_en216 := tonslide1.Q;
IF _en216 THEN _t216 := FALSE; END_IF;
_t218 := (speedImpuls4 = TRUE) OR _t221;
tonslide1(IN := _t212, PT := T#30s);
_t221 := speedImpuls4 = FALSE;
IF _en216 THEN run4 := _t216; END_IF;
dozSlide4 := tonslide1.Q;
END_PROGRAM

(* POU sinxron, ST *)
PROGRAM sinxron
VAR
	GetTime: CurTimeEx;
	TDate: SystemTimeDate;
	Sys_Time: SysTime64;
	need_day : UINT;
END_VAR
TDate.Day :=0;
TDate.DayOfWeek :=0;
TDate.dwHighMsec :=0;
TDate.dwLowMSecs :=0;
TDate.Milliseconds :=0;
TDate.Minute :=0;
TDate.Second :=0;
TDate.Hour :=0;
TDate.Year :=0;
TDate.Month :=0;
Sys_time.ulHigh :=0;
Sys_time.ulLow :=0;
GetTime (SystemTime:=Sys_Time , TimeDate:= TDate);
IF (timeSinxron = TRUE) THEN
	IF (minute <> 0) THEN
		TDate.Minute:=minute;
	END_IF;
	IF (sekund <>0) THEN
		TDate.Second:=sekund;
	END_IF;
	IF (hour <> 0) THEN
		TDate.Hour:=hour;
	END_IF;
	IF (day <> 0) THEN
		TDate.Day:=day;
	END_IF;
	IF (month <> 0) THEN
		TDate.Month:=month;
	END_IF;
	IF (year <> 0) THEN
		TDate.Year:=year;
	END_IF;
	GetTime (SystemTime:=Sys_Time , TimeDate:= TDate);
	timeSinxron := FALSE;
END_IF;
CASE TDate.Month OF
	1, 3, 5, 7, 8, 10, 12 : need_day := 31; (*Agar 1, 3, .. 12 oy lar bulsa 31 kuni hisoblagichni nolqilish*)
	2 : IF (TDate.Year MOD 4  = 0 AND TDate.Year MOD 100 > 0 OR TDate.Year MOD 400 = 0) THEN
			need_day := 29;  (*Agar yil kabisa yili  bulsa 29 kuni hisoblagichni nolqilish*)
		ELSE
			need_day := 28;  (*Agar yil kabisa yili EMAS bulsa 29 kuni hisoblagichni nolqilish*)
		END_IF;
	4, 6, 9, 11 : need_day := 30; (*Qolgan oylarda 30 kuni nol qilish*)
END_CASE;
END_PROGRAM

(* POU sirenStart, CFC *)
PROGRAM sirenStart
VAR
	tpStart: TP;
	blnk: BLINK;
	zvon: BOOL;
	trig: F_TRIG;
END_VAR
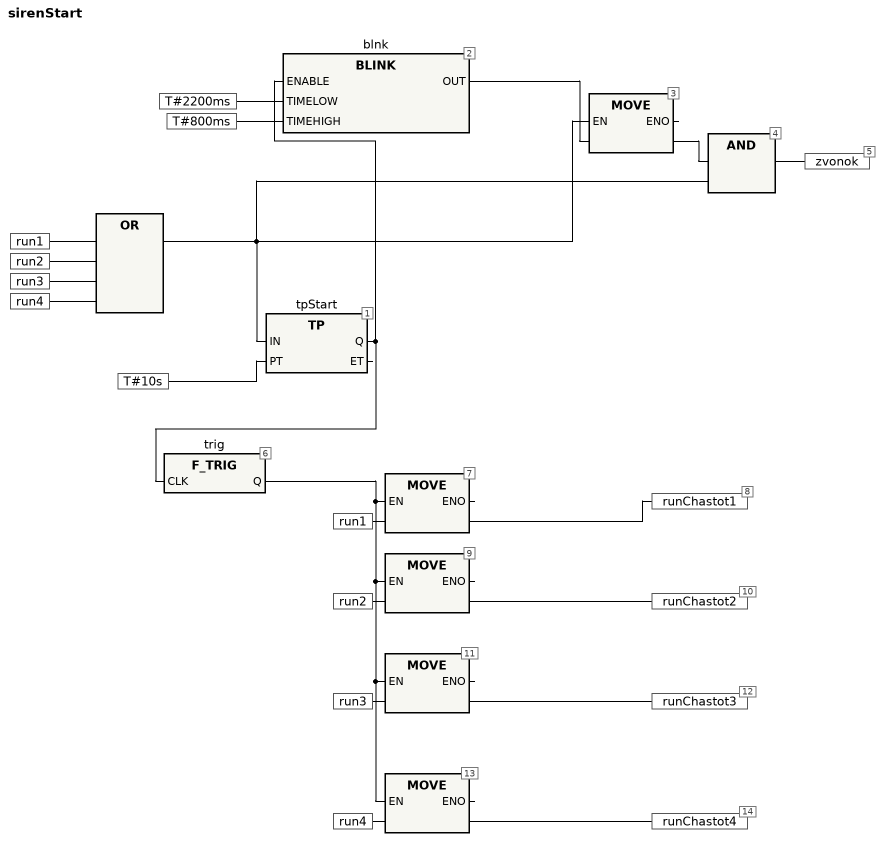
_CFC_ (* Continuous Function Chart, elements in execution order *)
#0 OR(run1, run2, run3, run4)
#1 tpStart:TP(IN: #0, PT: T#10s)
#2 blnk:BLINK(ENABLE: #1.Q, TIMELOW: T#2200ms, TIMEHIGH: T#800ms)
#3 MOVE(EN: #0, #2.OUT)
#4 AND(#3, #0)
#5 zvonok <= #4
#6 trig:F_TRIG(CLK: #1.Q)
#7 MOVE(EN: #6.Q, run1)
#8 runChastot1 <= #7
#9 MOVE(EN: #6.Q, run2)
#10 runChastot2 <= #9
#11 MOVE(EN: #6.Q, run3)
#12 runChastot3 <= #11
#13 MOVE(EN: #6.Q, run4)
#14 runChastot4 <= #13
_END_CFC_
END_PROGRAM

(* POU sirenStop, CFC *)
PROGRAM sirenStop
VAR
	tpStop: TP;
	zvon: BOOL;
	trig: R_TRIG;
	firstTime: BOOL;
END_VAR
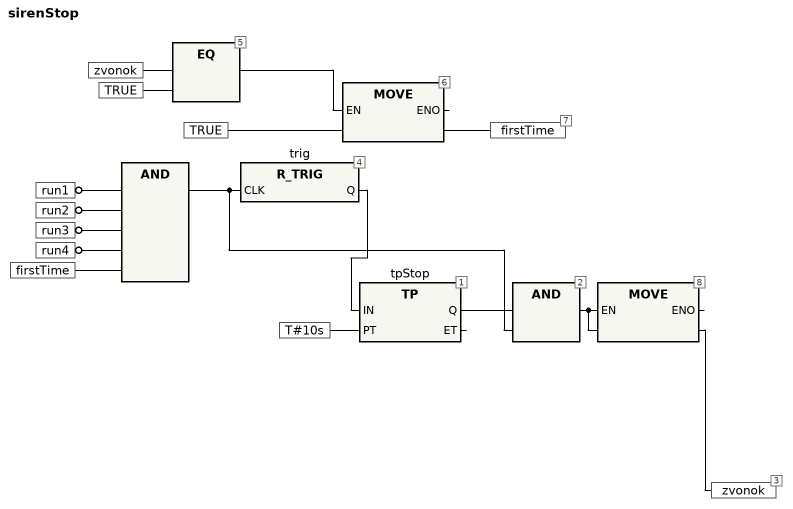
_CFC_ (* Continuous Function Chart, elements in execution order *)
#0 AND(NOT run1, NOT run2, NOT run3, NOT run4, firstTime)
#1 tpStop:TP(IN: #4.Q, PT: T#10s)
#2 AND(#1.Q, #0)
#3 zvonok <= #8
#4 trig:R_TRIG(CLK: #0)
#5 EQ(zvonok, TRUE)
#6 MOVE(EN: #5, TRUE)
#7 firstTime <= #6
#8 MOVE(EN: #2, #2)
_END_CFC_
END_PROGRAM

(* POU stopCFC, CFC *)
PROGRAM stopCFC
VAR
	fl_to_str1 : float_to_str;
	fl_to_str2 : float_to_str;
	fl_to_str3 : float_to_str;
	fl_to_str4 : float_to_str;
END_VAR
VAR (* helpers for the ST form of the networks *)
	_t1 : BOOL;
	_en30 : BOOL;
	_t30 : BOOL;
	_t6 : BOOL;
	_en32 : BOOL;
	_t32 : BOOL;
	_t10 : BOOL;
	_t35 : BOOL;
	_t14 : BOOL;
	_t37 : BOOL;
	_en65 : BOOL;
	_t65 : BOOL;
END_VAR
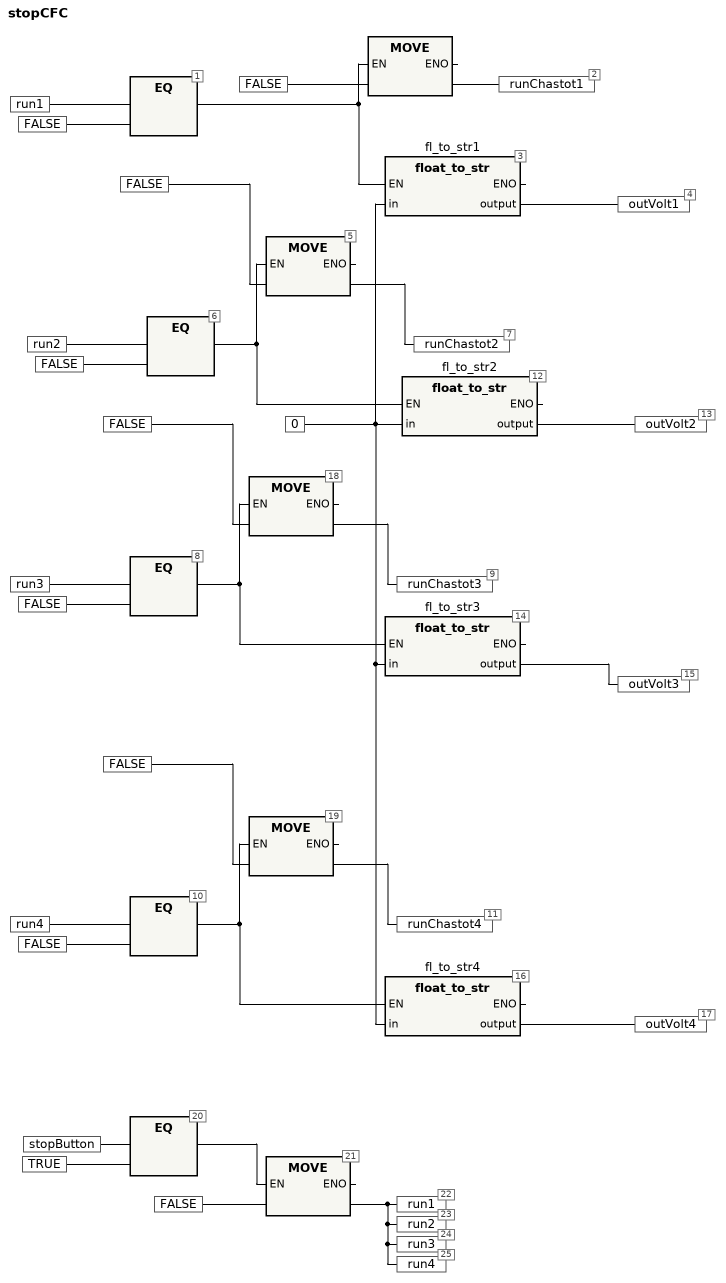
_CFC_ (* Continuous Function Chart, elements in execution order *)
#0 MOVE(EN: #1, FALSE)
#1 EQ(run1, FALSE)
#2 runChastot1 <= #0
#3 fl_to_str1:float_to_str(EN: #1, in: 0)
#4 outVolt1 <= #3.output
#5 MOVE(EN: #6, FALSE)
#6 EQ(run2, FALSE)
#7 runChastot2 <= #5
#8 EQ(run3, FALSE)
#9 runChastot3 <= #18
#10 EQ(run4, FALSE)
#11 runChastot4 <= #19
#12 fl_to_str2:float_to_str(EN: #6, in: 0)
#13 outVolt2 <= #12.output
#14 fl_to_str3:float_to_str(EN: #8, in: 0)
#15 outVolt3 <= #14.output
#16 fl_to_str4:float_to_str(EN: #10, in: 0)
#17 outVolt4 <= #16.output
#18 MOVE(EN: #8, FALSE)
#19 MOVE(EN: #10, FALSE)
#20 EQ(stopButton, TRUE)
#21 MOVE(EN: #20, FALSE)
#22 run1 <= #21
#23 run2 <= #21
#24 run3 <= #21
#25 run4 <= #21
_END_CFC_
(* the same logic as Structured Text *)
_en30 := _t1;
IF _en30 THEN _t30 := FALSE; END_IF;
_t1 := run1 = FALSE;
IF _en30 THEN runChastot1 := _t30; END_IF;
IF _t1 THEN fl_to_str1(in := 0); END_IF;
outVolt1 := fl_to_str1.output;
_en32 := _t6;
IF _en32 THEN _t32 := FALSE; END_IF;
_t6 := run2 = FALSE;
IF _en32 THEN runChastot2 := _t32; END_IF;
_t10 := run3 = FALSE;
runChastot3 := _t35;
_t14 := run4 = FALSE;
runChastot4 := _t37;
IF _t6 THEN fl_to_str2(in := 0); END_IF;
outVolt2 := fl_to_str2.output;
IF _t10 THEN fl_to_str3(in := 0); END_IF;
outVolt3 := fl_to_str3.output;
IF _t14 THEN fl_to_str4(in := 0); END_IF;
outVolt4 := fl_to_str4.output;
IF _t10 THEN _t35 := FALSE; END_IF;
IF _t14 THEN _t37 := FALSE; END_IF;
_en65 := stopButton = TRUE;
IF _en65 THEN _t65 := FALSE; END_IF;
IF _en65 THEN run1 := _t65; END_IF;
IF _en65 THEN run2 := _t65; END_IF;
IF _en65 THEN run3 := _t65; END_IF;
IF _en65 THEN run4 := _t65; END_IF;
END_PROGRAM

(* POU float_to_str, ST *)
FUNCTION_BLOCK float_to_str
VAR_INPUT
	in : REAL; (*Kiritiladigan son*)
END_VAR
VAR_OUTPUT
	output : STRING; (*tayyor konvertattsiya qilingan son*)
END_VAR
VAR
	butun : WORD;
	kasr: WORD;
	res : REAL;
	result : DWORD;
	lntrafo : LIN_TRAFO;
	input : REAL;
END_VAR
lntrafo(IN_MAX := 0, IN := LIMIT(0, in, 100) , IN_MAX := 100, OUT_MIN := 0, OUT_MAX := 10, OUT => input);

res :=input*1000;
result := REAL_TO_DWORD(res);
butun :=DWORD_TO_WORD( result / 1000);
kasr := DWORD_TO_WORD(result MOD 1000);
IF(butun< 10) THEN
	output := CONCAT(CONCAT(CONCAT('+', '0'),WORD_TO_STRING(butun)) , '.' );
ELSE
	output := CONCAT(CONCAT('+', WORD_TO_STRING(butun)) , '.' );
END_IF;
IF(kasr = 0) THEN
	output := CONCAT(output, '000');
ELSE
	output := CONCAT(output, WORD_TO_STRING(kasr));
END_IF
END_FUNCTION_BLOCK

(* POU taraSpeedModeDoz1, ST *)
PROGRAM taraSpeedModeDoz1
VAR
	fls : float_to_str;
	statist : STATISTICS_REAL;
	chastot : FREQ_MEASURE;
	trig : R_TRIG;
END_VAR
(**********************************************************)
fls(in := WORD_TO_REAL(taskDozSpeed1), output => outVolt1);
IF (KoefSpeed1 = TRUE) THEN
	dozKoefSpeedDoz1 := taraSpeedDoz1 / freqChastot1;
END_IF;
(**********************************************************)
END_PROGRAM

(* POU taraSpeedModeDoz2, ST *)
PROGRAM taraSpeedModeDoz2
VAR
	fls : float_to_str;
	statist : STATISTICS_REAL;
	chastot : FREQ_MEASURE;
	trig : R_TRIG;
END_VAR
(**********************************************************)
fls(in := WORD_TO_REAL(taskDozSpeed2), output => outVolt2);
IF (KoefSpeed2 = TRUE) THEN
	dozKoefSpeedDoz2 := taraSpeedDoz2 / freqChastot2;
END_IF;
(**********************************************************)
END_PROGRAM

(* POU taraSpeedModeDoz3, ST *)
PROGRAM taraSpeedModeDoz3
VAR
	fls : float_to_str;
	statist : STATISTICS_REAL;
	chastot : FREQ_MEASURE;
	trig : R_TRIG;
END_VAR
(**********************************************************)
fls(in := WORD_TO_REAL(taskDozSpeed3), output => outVolt3);
IF (KoefSpeed3 = TRUE) THEN
	dozKoefSpeedDoz3 := taraSpeedDoz3 / freqChastot3;
END_IF;
(**********************************************************)
END_PROGRAM

(* POU taraSpeedModeDoz4, ST *)
PROGRAM taraSpeedModeDoz4
VAR
	fls : float_to_str;
	statist : STATISTICS_REAL;
	chastot : FREQ_MEASURE;
	trig : R_TRIG;
END_VAR
(**********************************************************)
fls(in := WORD_TO_REAL(taskDozSpeed4), output => outVolt4);
IF (KoefSpeed4 = TRUE) THEN
	dozKoefSpeedDoz4 := taraSpeedDoz4 / freqChastot4;
END_IF;
(**********************************************************)
END_PROGRAM

(* POU taraVesModeDoz1, ST *)
PROGRAM taraVesModeDoz1
VAR
	fls : float_to_str;
	statist : STATISTICS_REAL;
	chastot : FREQ_MEASURE;
	trig : R_TRIG;
END_VAR
(**********************************************************)
IF (dreyf1 = TRUE) THEN
	dozDreyfDoz1 :=
	dozMilliVolt1;
END_IF;
IF (KoefPer1 = TRUE) THEN
	dozKoefPerVESDoz1 :=
	taraVesDoz1 / (dozMilliVolt1 -
	dozDreyfDoz1);
END_IF;

(**********************************************************)
END_PROGRAM

(* POU taraVesModeDoz2, ST *)
PROGRAM taraVesModeDoz2
VAR
	fls : float_to_str;
	statist : STATISTICS_REAL;
	chastot : FREQ_MEASURE;
	trig : R_TRIG;
END_VAR
(**********************************************************)
IF (dreyf2 = TRUE) THEN
	dozDreyfDoz2 :=
	dozMilliVolt2;
END_IF;
IF (KoefPer2 = TRUE) THEN
	dozKoefPerVESDoz2 :=
	taraVesDoz2 / (dozMilliVolt2 -
	dozDreyfDoz2);
END_IF;

(**********************************************************)
END_PROGRAM

(* POU taraVesModeDoz3, ST *)
PROGRAM taraVesModeDoz3
VAR
	fls : float_to_str;
	statist : STATISTICS_REAL;
	chastot : FREQ_MEASURE;
	trig : R_TRIG;
END_VAR
(**********************************************************)
IF (dreyf3 = TRUE) THEN
	dozDreyfDoz3 :=
	dozMilliVolt3;
END_IF;
IF (KoefPer3 = TRUE) THEN
	dozKoefPerVESDoz3 :=
	taraVesDoz1 / (dozMilliVolt3 -
	dozDreyfDoz3);
END_IF;

(**********************************************************)
END_PROGRAM

(* POU taraVesModeDoz4, ST *)
PROGRAM taraVesModeDoz4
VAR
	fls : float_to_str;
	statist : STATISTICS_REAL;
	chastot : FREQ_MEASURE;
	trig : R_TRIG;
END_VAR
(**********************************************************)
IF (dreyf4 = TRUE) THEN
	dozDreyfDoz4 :=
	dozMilliVolt4;
END_IF;
IF (KoefPer4 = TRUE) THEN
	dozKoefPerVESDoz4 :=
	taraVesDoz4 / (dozMilliVolt4 -
	dozDreyfDoz4);
END_IF;

(**********************************************************)
END_PROGRAM

(* POU auto, CFC *)
PROGRAM auto
VAR
	doz1: dozator;
	doz2: dozator;
	doz3: dozator;
	doz4: dozator;
	fltstr1: float_to_str;
	fltstr2: float_to_str;
	fltstr3: float_to_str;
	fltstr4: float_to_str;

END_VAR
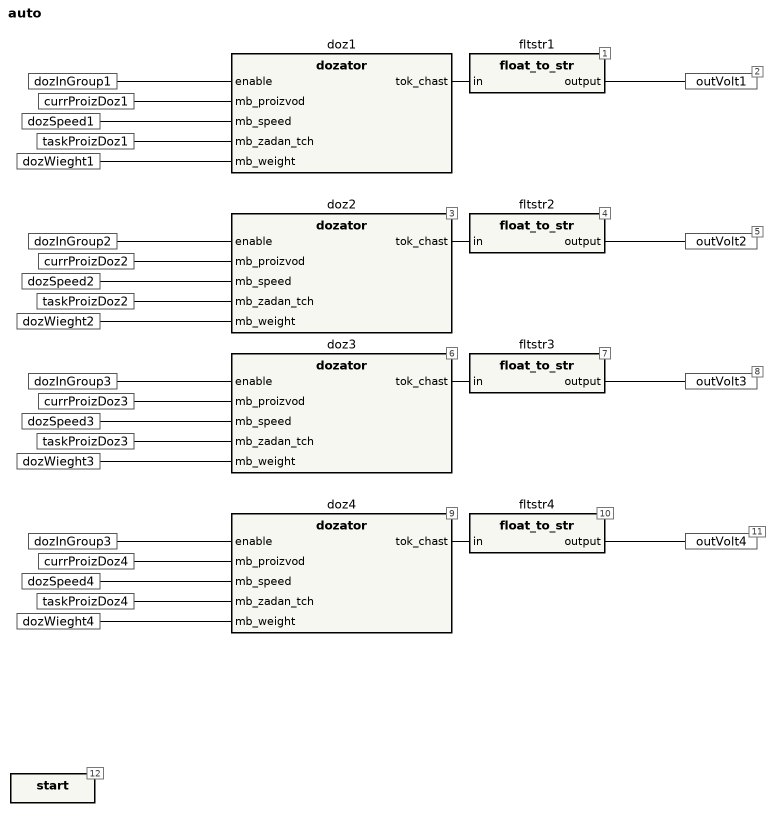
_CFC_ (* Continuous Function Chart, elements in execution order *)
#0 doz1:dozator(enable: dozInGroup1, mb_proizvod: currProizDoz1, mb_speed: dozSpeed1, mb_zadan_tch: taskProizDoz1, mb_weight: dozWieght1)
#1 fltstr1:float_to_str(in: #0.tok_chast)
#2 outVolt1 <= #1.output
#3 doz2:dozator(enable: dozInGroup2, mb_proizvod: currProizDoz2, mb_speed: dozSpeed2, mb_zadan_tch: taskProizDoz2, mb_weight: dozWieght2)
#4 fltstr2:float_to_str(in: #3.tok_chast)
#5 outVolt2 <= #4.output
#6 doz3:dozator(enable: dozInGroup3, mb_proizvod: currProizDoz3, mb_speed: dozSpeed3, mb_zadan_tch: taskProizDoz3, mb_weight: dozWieght3)
#7 fltstr3:float_to_str(in: #6.tok_chast)
#8 outVolt3 <= #7.output
#9 doz4:dozator(enable: dozInGroup3, mb_proizvod: currProizDoz4, mb_speed: dozSpeed4, mb_zadan_tch: taskProizDoz4, mb_weight: dozWieght4)
#10 fltstr4:float_to_str(in: #9.tok_chast)
#11 outVolt4 <= #10.output
#12 start()
_END_CFC_
(* the same logic as Structured Text *)
doz1(enable := dozInGroup1, mb_proizvod := currProizDoz1, mb_speed := dozSpeed1, mb_zadan_tch := taskProizDoz1, mb_weight := dozWieght1);
fltstr1(in := doz1.tok_chast);
outVolt1 := fltstr1.output;
doz2(enable := dozInGroup2, mb_proizvod := currProizDoz2, mb_speed := dozSpeed2, mb_zadan_tch := taskProizDoz2, mb_weight := dozWieght2);
fltstr2(in := doz2.tok_chast);
outVolt2 := fltstr2.output;
doz3(enable := dozInGroup3, mb_proizvod := currProizDoz3, mb_speed := dozSpeed3, mb_zadan_tch := taskProizDoz3, mb_weight := dozWieght3);
fltstr3(in := doz3.tok_chast);
outVolt3 := fltstr3.output;
doz4(enable := dozInGroup3, mb_proizvod := currProizDoz4, mb_speed := dozSpeed4, mb_zadan_tch := taskProizDoz4, mb_weight := dozWieght4);
fltstr4(in := doz4.tok_chast);
outVolt4 := fltstr4.output;
start();
END_PROGRAM

(* POU dozator, ST *)
FUNCTION_BLOCK dozator
VAR_INPUT
	enable : BOOL;
	mb_proizvod: REAL;
	mb_speed: REAL;
	mb_zadan_tch: REAL;
	mb_weight: REAL;
END_VAR
VAR_OUTPUT
	tok_chast : REAL;

END_VAR
VAR
	tmr_t : TON;
	tmp_tok_chast: REAL;
	old_tok_chast: REAL;
	old_weight: REAL;
	mahraj: REAL;
	old_speed: REAL;
	surat: REAL;
	tError : TON;
END_VAR
IF(enable = TRUE) THEN
	tmr_t(in := TRUE, pt := t#1000ms);

	IF (tmr_t.Q = TRUE) THEN
	old_tok_chast := tok_chast;
	old_speed := mb_speed;

	mb_proizvod := (old_weight *
					 mb_speed * 36)/1000; (* 45 = 3600 cek / 80 cm *)

	IF (old_weight > 0) THEN
		(*tok_chast := ((tok_chast - 4) * mb_zadan_tch *1000) / (45 * old_weight * mb_speed) + 4;*)
		surat := (old_tok_chast) *
					mb_zadan_tch * 1000;
		mahraj := (36 * old_weight *
				mb_speed);
		tmp_tok_chast := (surat /mahraj );

		IF((tmp_tok_chast - old_tok_chast) > 0.5) THEN
			tmp_tok_chast := old_tok_chast + 0.5;
		END_IF;
		IF((tmp_tok_chast - old_tok_chast) < 0.5) THEN
			tmp_tok_chast := old_tok_chast - 0.5;
		END_IF;
		IF (tmp_tok_chast < 0) THEN
			tmp_tok_chast := 0;
		END_IF;
		IF (tmp_tok_chast > 100) THEN
			tmp_tok_chast := 100;
		END_IF;
			tok_chast := tmp_tok_chast;
			old_weight := mb_weight;
	ELSE
		tmp_tok_chast := 25;
		old_weight := mb_weight;
	END_IF;
	tmr_t(in := FALSE);
	END_IF;
ELSE
	tok_chast := 0;
END_IF;
(*
tError(in := mb_weight < 5 AND NOT resetError, PT := T#15s);
IF(tError.Q = TRUE) THEN
	error := TRUE;
	tok_chast := 0;
END_IF;
IF (resetError = TRUE) THEN
	error := FALSE;
	reset := FALSE;
	tError(in := FALSE);
END_IF;
*)
END_FUNCTION_BLOCK

(* POU start, ST *)
PROGRAM start
VAR
END_VAR
(*
run1 := dozAuto1 AND dozInGroup1;
run2 := dozAuto2 AND dozInGroup2;
run3 := dozAuto3 AND dozInGroup3;
run4 := dozAuto4 AND dozInGroup4;
*);
IF (dozInGroup1 = FALSE) THEN
	run1 := FALSE;
END_IF;
IF (dozInGroup2 = FALSE) THEN
	run2 := FALSE;
END_IF;
IF (dozInGroup3 = FALSE) THEN
	run3 := FALSE;
END_IF;
IF (dozInGroup4 = FALSE) THEN
	run4 := FALSE;
END_IF;
IF(starButton = TRUE)THEN
	run1 := TRUE;
	run2 := TRUE;
	run3 := TRUE;
	run4 := TRUE;
END_IF;
END_PROGRAM

(* POU calc_time, CFC *)
FUNCTION_BLOCK calc_time
VAR_INPUT
	impuls: BOOL;
END_VAR
VAR_OUTPUT
	totalTime : UINT;
END_VAR
VAR
	rtirg1: R_TRIG;
	ton1: TON;
	res: BOOL;
	ftirg1: F_TRIG;
	tp1: TP;
	strt_ton: BOOL;
END_VAR
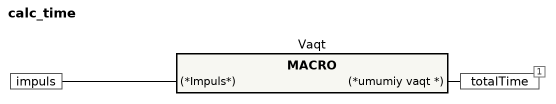
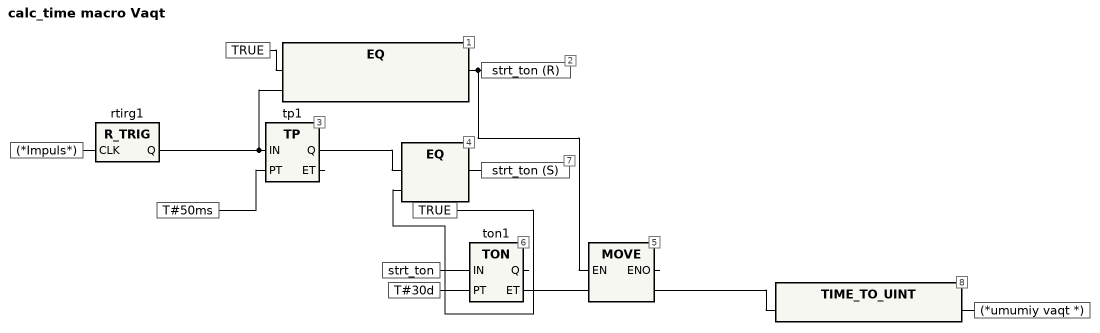
_CFC_ (* Continuous Function Chart, elements in execution order *)
#0 MACRO Vaqt(pin 1 "(*Impuls*)": impuls)
	#1 rtirg1:R_TRIG(CLK: pin 1)
	#2 EQ(TRUE, #1.Q)
	#3 R strt_ton <= #2
	#4 tp1:TP(IN: #1.Q, PT: T#50ms)
	#5 EQ(#4.Q, TRUE)
	#6 MOVE(EN: #2, #7.ET)
	#7 ton1:TON(IN: strt_ton, PT: T#30d)
	#8 S strt_ton <= #5
	out 1 "(*umumiy vaqt *)" <= #9
	#9 TIME_TO_UINT(#6)
END_MACRO
#10 totalTime <= #0.out 1
_END_CFC_
END_FUNCTION_BLOCK
